CASE Phase OF
	0:
		Inner.SetLabel('CHAR_Timeout_Subject');
		Inner.AddReporter(Recorder);
		Defaults.Body.Cycles	  := 5;
		Defaults.Body.IsCyclesSet := TRUE;
		Inner.SetDefaults(Defaults);

		// Claims nothing: inherits both units from the suite.
		Inner.Register(DefaultCycles, 'DefaultCycles', Budgets);

		// Claims its own scan budget.
		OwnCycles.Body.Cycles	   := 20;
		OwnCycles.Body.IsCyclesSet := TRUE;
		Inner.Register(OverrideCycles, 'OverrideCycles', OwnCycles);

		// Claims the wall clock ONLY, and long enough that it cannot be what fires.

		// The suite's five-cycle budget must still end this test.
		OwnTimeOnly.Body.Timeout	  := T#10S;
		OwnTimeOnly.Body.IsTimeoutSet := TRUE;
		Inner.Register(OverrideTimeOnly, 'OverrideTimeOnly', OwnTimeOnly);
		Phase := 1;
		Run	  := FALSE;

	1:
		IF Inner.Run(Enable := TRUE) THEN
			Phase := 2;
		END_IF

		Run := FALSE;

	2:
		ExpectedCount := 3;
		ActualCount	  := Recorder.StatFailures;
		Test.AssertEqual(ExpectedCount, ActualCount, 'all three hit a deadline');
		Test.AssertTrue(Recorder.FailureContains('DefaultCycles', 'after 5 cycles'), 'suite default applies when nothing was claimed');
		Test.AssertTrue(Recorder.FailureContains('OverrideCycles', 'after 20 cycles'), 'the per-test cycle budget wins');

		// The subtle one.
		Test.AssertTrue(Recorder.FailureContains('OverrideTimeOnly', 'after 5 cycles'), 'claiming the wall clock leaves the cycle budget inherited');

		// And each really ran for its own budget, not somebody else's.
		ExpectedCount := 5;
		ActualCount	  := DefaultCycles.BodyCalls;
		Test.AssertEqual(ExpectedCount, ActualCount, 'the default test ran five scans');
		ExpectedCount := 20;
		ActualCount	  := OverrideCycles.BodyCalls;
		Test.AssertEqual(ExpectedCount, ActualCount, 'the overriding test ran twenty');
		Run := TRUE;
END_CASE
END_METHOD

END_FUNCTION_BLOCK

// ---- Tests/Characterization/CHAR_SerialExecution.TcPOU
// Part of the acceptance contract: no test body runs while another is running.

//

// Tests share the scan and usually share fixtures, so predictable and slow beats

// fast and flaky. Serial execution is structural here - the arbiter hands out one

// test and the runner drives one - so this is a guard against a future change

// rather than a check on today's code, and it would be caught here and nowhere

// else.

//

// A test cannot observe this about another test: it is handed nothing but its own

// assertion handle. So the tests report in and out of a shared witness and the

// contract becomes one number, MaxConcurrent. TotalEntries stops that number being

// satisfied by nothing running at all.
FUNCTION_BLOCK CHAR_SerialExecution IMPLEMENTS I_Test
VAR
	Inner			   : TestSuite<4>;
	Recorder		   : RecordingReporter;
	Budgets			   : ST_TestBudgets;
	Phase			   : DINT;
	Scans			   : DINT;
	Witness			   : ConcurrencyWitness;
	Long			   : WitnessedTest;
	Second			   : WitnessedTest;
	Third			   : WitnessedTest;
	ExpectedConcurrent : DINT;
	ActualConcurrent   : DINT;
	ExpectedEntries	   : DINT;
	ActualEntries	   : DINT;
	ExpectedCount	   : UDINT;
	ActualCount		   : UDINT;
END_VAR

METHOD Run : BOOL
VAR_INPUT
	Enable : BOOL;
	Test   : I_TestAssertions;
END_VAR
Scans := Scans + 1;
IF Scans > 500 THEN
	Test.Fail('the inner suite never completed');
	Run := TRUE;
	RETURN;
END_IF

CASE Phase OF
	0:
		Inner.SetLabel('CHAR_Serial_Subject');
		Inner.AddReporter(Recorder);

		// Multi-scan deliberately: a single-scan test could never overlap anything, so

		// a suite of them would prove this by accident rather than by design.
		Long.Attach(Scans := 8, Witness := Witness);
		Second.Attach(Scans := 4, Witness := Witness);
		Third.Attach(Scans := 4, Witness := Witness);
		Inner.Register(Long, 'Long', Budgets);
		Inner.Register(Second, 'Second', Budgets);
		Inner.Register(Third, 'Third', Budgets);
		Phase := 1;
		Run	  := FALSE;

	1:
		IF Inner.Run(Enable := TRUE) THEN
			Phase := 2;
		END_IF

		Run := FALSE;

	2:
		ExpectedConcurrent := 1;
		ActualConcurrent   := Witness.MaxConcurrent;
		Test.AssertEqual(ExpectedConcurrent, ActualConcurrent, 'no test body ran while another was running');

		// Without this, nothing running at all would satisfy the line above.
		ExpectedEntries := 3;
		ActualEntries	:= Witness.TotalEntries;
		Test.AssertEqual(ExpectedEntries, ActualEntries, 'and all three really ran');
		ExpectedCount := 3;
		ActualCount	  := Recorder.StatTests;
		Test.AssertEqual(ExpectedCount, ActualCount, 'all three were registered');
		ExpectedCount := 0;
		ActualCount	  := Recorder.StatFailures;
		Test.AssertEqual(ExpectedCount, ActualCount, 'and all three passed');
		Run := TRUE;
END_CASE
END_METHOD

END_FUNCTION_BLOCK

// ---- Doubles/ConcurrencyWitness.TcPOU
// Counts how many tests are inside their body at the same moment.

//

// A test cannot observe this about another test - it is handed nothing but its own

// assertion handle, which is the founding constraint working as intended.

//

// So tests report in and out of a shared witness instead, and the contract becomes

// one number: MaxConcurrent must never exceed 1.
FUNCTION_BLOCK ConcurrencyWitness
VAR
	_Active		   : DINT;
	_MaxConcurrent : DINT;
	_TotalEntries  : DINT;
END_VAR

// A test body has started. Called on its FIRST scan only.
METHOD Enter
_Active		  := _Active + 1;
_TotalEntries := _TotalEntries + 1;
IF _Active > _MaxConcurrent THEN
	_MaxConcurrent := _Active;
END_IF
END_METHOD

// A test body has finished. Called on its LAST scan only.
METHOD Leave
_Active := _Active - 1;
END_METHOD

// The most tests ever inside a body at once. Must be 1: tests share the scan and

// usually share fixtures, so predictable and slow beats fast and flaky.
PROPERTY MaxConcurrent : DINT
GET
MaxConcurrent := _MaxConcurrent;
END_GET
END_PROPERTY

METHOD Reset
_Active		   := 0;
_MaxConcurrent := 0;
_TotalEntries  := 0;
END_METHOD

// How many bodies started. Proves every test really ran, so a MaxConcurrent of 1

// cannot be achieved by nothing running at all.
PROPERTY TotalEntries : DINT
GET
TotalEntries := _TotalEntries;
END_GET
END_PROPERTY

END_FUNCTION_BLOCK

// ---- Doubles/WitnessedTest.TcPOU
// A multi-scan test that reports its entry and exit to a shared witness.

//

// Takes several scans deliberately: a single-scan test could never overlap

// anything, so a suite of them would prove serial execution by accident rather

// than by design.
FUNCTION_BLOCK WitnessedTest IMPLEMENTS I_Test
VAR
	// A REFERENCE TO, not an instance: every test in the suite must report to the

	// SAME witness, or each would see itself alone and MaxConcurrent would be 1 by

	// construction rather than by the suite behaving.
	_Witness	: REFERENCE TO ConcurrencyWitness;
	_Scans		: UDINT := 4;
	_Calls		: UDINT;
	_HasEntered : BOOL;
END_VAR

// The shared witness, and how many scans this test should take.
METHOD Attach
VAR_INPUT
	Scans : UDINT;
END_VAR

VAR_IN_OUT
	Witness : ConcurrencyWitness;
END_VAR
_Witness REF= Witness;
_Scans	 := Scans;
END_METHOD

METHOD Run : BOOL
VAR_INPUT
	Enable : BOOL;
	Test   : I_TestAssertions;
END_VAR
IF NOT Enable THEN
	Run := TRUE;
	RETURN;
END_IF

IF NOT __ISVALIDREF(_Witness) THEN
	Test.ReportError('no witness was attached');
	Run := TRUE;
	RETURN;
END_IF

IF NOT _HasEntered THEN
	_HasEntered := TRUE;
	_Witness.Enter();
END_IF

_Calls := _Calls + 1;
IF _Calls < _Scans THEN
	Run := FALSE;
	RETURN;
END_IF

Test.AssertTrue(TRUE, 'ran to completion');
_Witness.Leave();
Run := TRUE;
END_METHOD

END_FUNCTION_BLOCK
